// TIA Portal V16 export
// export: Created 2022-09-01T13:36:55.5389908Z, ExportSetting WithDefaults, DisplayName Totally Integrated Automation Portal, DisplayVersion V16, DisplayName TIA Portal Version Control Interface, DisplayVersion V16, DisplayName TIA Portal Openness, DisplayVersion V16, DisplayName STEP 7 Professional, DisplayVersion V16, DisplayName STEP 7 Safety, DisplayVersion V16, DisplayName WinCC Advanced, DisplayVersion V16
FUNCTION "Alim_Processo" : Void   // FC1, LAD
{ S7_Optimized_Access := 'TRUE' }
VERSION : 0.1
// stored: AutoNumber true, IsIECCheckEnabled false, SetENOAutomatically false, UDAEnableTagReadback false
BEGIN

REGION Network 1: Etapa 10 (INÍCIO)
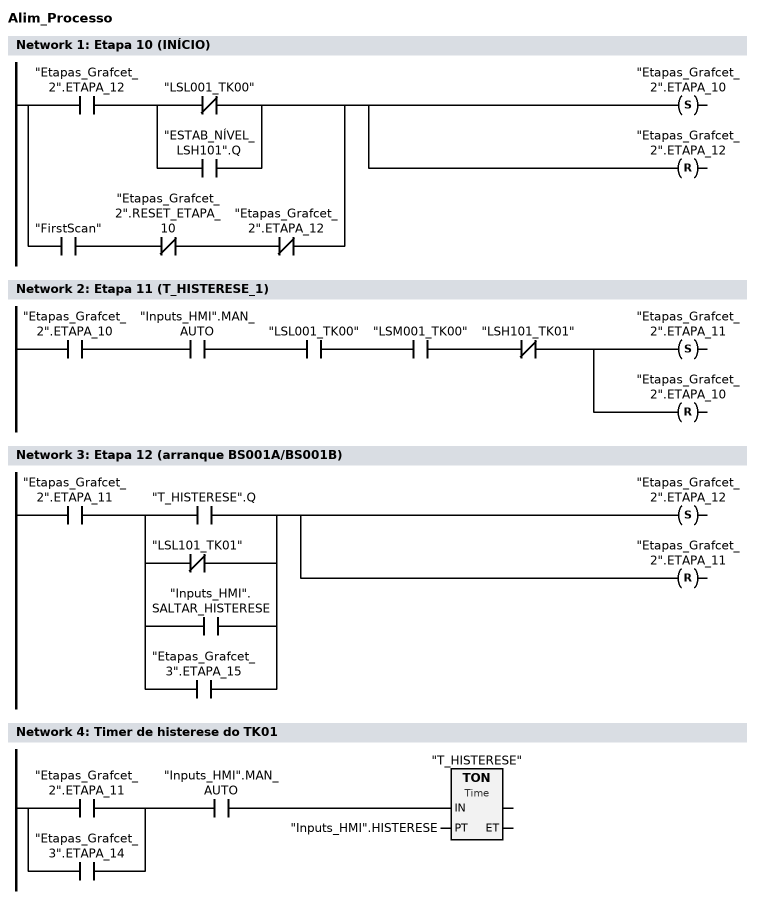
   RUNG wire#powerrail
      Contact( "Etapas_Grafcet_2".ETAPA_12 )
      wire#w1
      I_Contact( "LSL001_TK00" )
      wire#w2
      S_Coil( "Etapas_Grafcet_2".ETAPA_10 )
   END_RUNG
   RUNG wire#w1
      Contact( "ESTAB_NÍVEL_LSH101".Q )
   END_RUNG wire#w2
   RUNG wire#powerrail
      Contact( "FirstScan" )
      I_Contact( "Etapas_Grafcet_2".RESET_ETAPA_10 )
      I_Contact( "Etapas_Grafcet_2".ETAPA_12 )
   END_RUNG wire#w2
   RUNG wire#w2
      R_Coil( "Etapas_Grafcet_2".ETAPA_12 )
   END_RUNG
   // the same network as SCL:
   IF ("Etapas_Grafcet_2".ETAPA_12 AND (NOT "LSL001_TK00" OR "ESTAB_NÍVEL_LSH101".Q)) OR ("FirstScan" AND NOT "Etapas_Grafcet_2".RESET_ETAPA_10 AND NOT "Etapas_Grafcet_2".ETAPA_12) THEN
       "Etapas_Grafcet_2".ETAPA_10 := TRUE;
       "Etapas_Grafcet_2".ETAPA_12 := FALSE;
   END_IF;
END_REGION

REGION Network 2: Etapa 11 (T_HISTERESE_1)
   RUNG wire#powerrail
      Contact( "Etapas_Grafcet_2".ETAPA_10 )
      Contact( "Inputs_HMI".MAN_AUTO )
      Contact( "LSL001_TK00" )
      Contact( "LSM001_TK00" )
      I_Contact( "LSH101_TK01" )
      wire#w1
      S_Coil( "Etapas_Grafcet_2".ETAPA_11 )
   END_RUNG
   RUNG wire#w1
      R_Coil( "Etapas_Grafcet_2".ETAPA_10 )
   END_RUNG
   // the same network as SCL:
   IF "Etapas_Grafcet_2".ETAPA_10 AND "Inputs_HMI".MAN_AUTO AND "LSL001_TK00" AND "LSM001_TK00" AND NOT "LSH101_TK01" THEN
       "Etapas_Grafcet_2".ETAPA_11 := TRUE;
       "Etapas_Grafcet_2".ETAPA_10 := FALSE;
   END_IF;
END_REGION

REGION Network 3: Etapa 12 (arranque BS001A/BS001B)
   RUNG wire#powerrail
      Contact( "Etapas_Grafcet_2".ETAPA_11 )
      wire#w1
      Contact( "T_HISTERESE".Q )
      wire#w2
      S_Coil( "Etapas_Grafcet_2".ETAPA_12 )
   END_RUNG
   RUNG wire#w1
      I_Contact( "LSL101_TK01" )
   END_RUNG wire#w2
   RUNG wire#w1
      Contact( "Inputs_HMI".SALTAR_HISTERESE )
   END_RUNG wire#w2
   RUNG wire#w1
      Contact( "Etapas_Grafcet_3".ETAPA_15 )
   END_RUNG wire#w2
   RUNG wire#w2
      R_Coil( "Etapas_Grafcet_2".ETAPA_11 )
   END_RUNG
   // the same network as SCL:
   IF "Etapas_Grafcet_2".ETAPA_11 AND ("T_HISTERESE".Q OR NOT "LSL101_TK01" OR "Inputs_HMI".SALTAR_HISTERESE OR "Etapas_Grafcet_3".ETAPA_15) THEN
       "Etapas_Grafcet_2".ETAPA_12 := TRUE;
       "Etapas_Grafcet_2".ETAPA_11 := FALSE;
   END_IF;
END_REGION

REGION Network 4: Timer de histerese do TK01
   RUNG wire#powerrail
      Contact( "Etapas_Grafcet_2".ETAPA_11 )
      wire#w1
      Contact( "Inputs_HMI".MAN_AUTO )
      { S7_Templates := "time_type := Time" } "T_HISTERESE".TON(pt := "Inputs_HMI".HISTERESE, et =>)
   END_RUNG
   RUNG wire#powerrail
      Contact( "Etapas_Grafcet_3".ETAPA_14 )
   END_RUNG wire#w1
   // the same network as SCL:
   "T_HISTERESE".TON(IN := ("Etapas_Grafcet_2".ETAPA_11 OR "Etapas_Grafcet_3".ETAPA_14) AND "Inputs_HMI".MAN_AUTO,
                     PT := "Inputs_HMI".HISTERESE);
END_REGION
END_FUNCTION
